{attribute 'qualified_only'}
TYPE E_DrivingPinCtrl :
(
	Horizontal,
	Vertical
)USINT;
END_TYPE

(* stored: Version 1.1.0.1, ProductVersion 3.1.4024.11
   DUT E_DrivingPinCtrl: Id {eeb81d14-5d06-4001-9b66-e16c3c57137b} *)
